SUBAPPLICATION Uebung_043 (* Scaling Function Block with limits Testing *)
  (* Standard: 61499-2 *)
  (* Version 1.0, 2023-10-23, franz *)
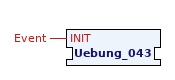
  EVENT_INPUT
    INIT;
  END_EVENT
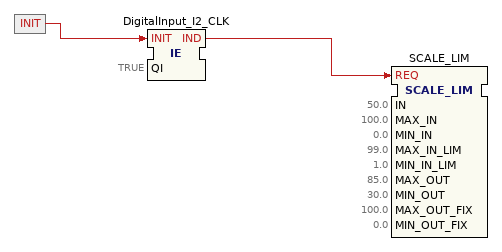
  FBS
    DigitalInput_I2_CLK : IE(QI := TRUE);
    SCALE_LIM : signalprocessing::SCALE_LIM(IN := 50.0, MAX_IN := 100.0, MIN_IN := 0.0, MAX_IN_LIM := 99.0, MIN_IN_LIM := 1.0, MAX_OUT := 85.0, MIN_OUT := 30.0, MAX_OUT_FIX := 100.0, MIN_OUT_FIX := 0.0);
  END_FBS
  EVENT_CONNECTIONS
    INIT TO DigitalInput_I2_CLK.INIT;
    DigitalInput_I2_CLK.IND TO SCALE_LIM.REQ;
  END_CONNECTIONS
END_SUBAPPLICATION
